Omron CX-Programmer project 新規ﾌﾟﾛｼﾞｪｸﾄ (CX-Programmer 9.61)

# PLC 新規PLC1: CP1L L

## Program 新規ﾌﾟﾛｸﾞﾗﾑ1 (cyclic task 0)

### Section ｾｸｼｮﾝ1

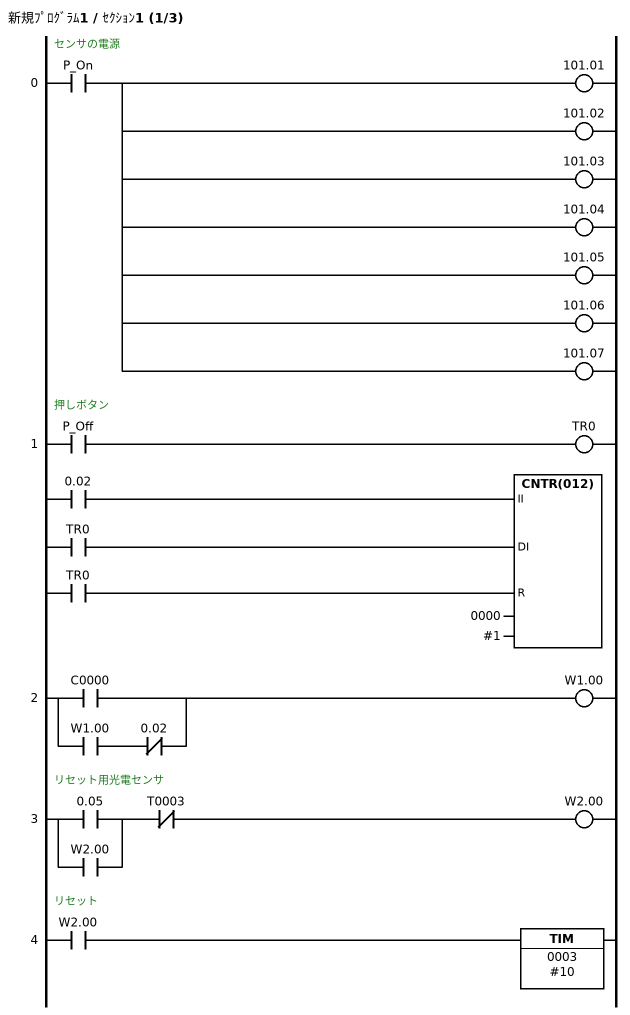
; rung 0: センサの電源
LD P_On
OUT 101.01
OUT 101.02
OUT 101.03
OUT 101.04
OUT 101.05
OUT 101.06
OUT 101.07
; rung 1: 押しボタン
LD 0.02
LD P_Off
OUT TR0
LD TR0
CNTR(012) 0000 #1
; rung 2
LD C0000
LD W1.00
ANDNOT 0.02
ORLD
OUT W1.00
; rung 3: リセット用光電センサ
LD 0.05
OR W2.00
ANDNOT T0003
OUT W2.00
; rung 4: リセット
LD W2.00
TIM 0003 #10

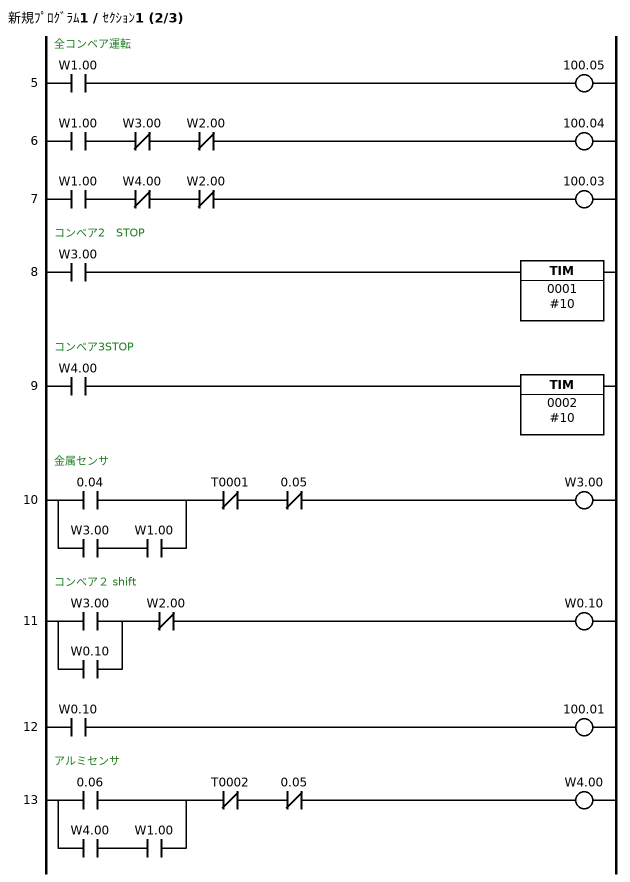
; rung 5: 全コンベア運転
LD W1.00
OUT 100.05
; rung 6
LD W1.00
ANDNOT W3.00
ANDNOT W2.00
OUT 100.04
; rung 7
LD W1.00
ANDNOT W4.00
ANDNOT W2.00
OUT 100.03
; rung 8: コンベア2　STOP
LD W3.00
TIM 0001 #10
; rung 9: コンベア3STOP
LD W4.00
TIM 0002 #10
; rung 10: 金属センサ
LD 0.04
LD W3.00
AND W1.00
ORLD
ANDNOT T0001
ANDNOT 0.05
OUT W3.00
; rung 11: コンベア２ shift
LD W3.00
OR W0.10
ANDNOT W2.00
OUT W0.10
; rung 12
LD W0.10
OUT 100.01
; rung 13: アルミセンサ
LD 0.06
LD W4.00
AND W1.00
ORLD
ANDNOT T0002
ANDNOT 0.05
OUT W4.00
; rung 14: コンベア3　shift

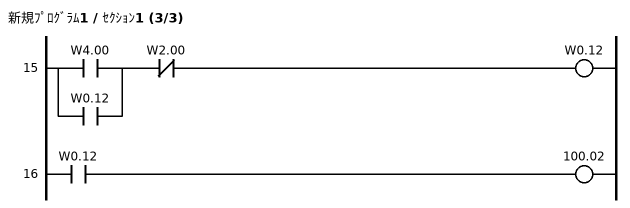
; rung 15
LD W4.00
OR W0.12
ANDNOT W2.00
OUT W0.12
; rung 16
LD W0.12
OUT 100.02

### Section END
; rung 0
END(001)